// Mitsubishi GX Works2 project: 실린더제어요약   PLC: Q02/Q02H

PROGRAM MAIN
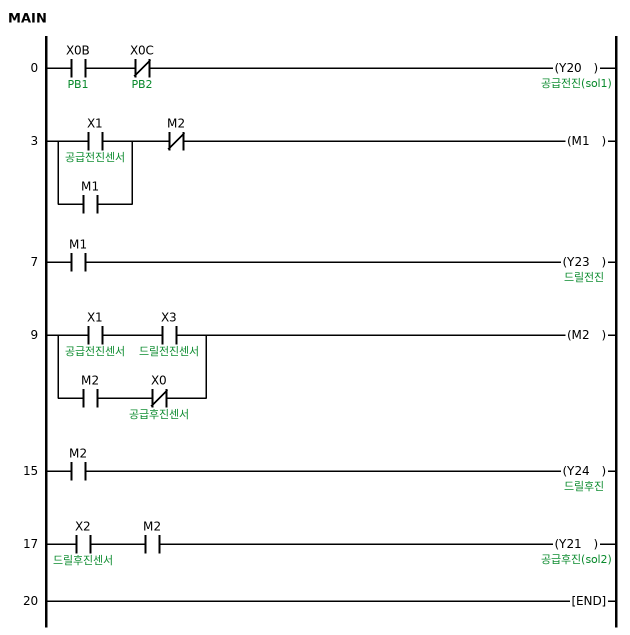
0     LD      X0B  ; PB1
      ANI     X0C  ; PB2
      OUT     Y20  ; 공급전진(sol1)
3     LD      X1  ; 공급전진센서
      OR      M1
      ANI     M2
      OUT     M1
7     LD      M1
      OUT     Y23  ; 드릴전진
9     LD      X1  ; 공급전진센서
      AND     X3  ; 드릴전진센서
      LD      M2
      ANI     X0  ; 공급후진센서
      ORB
      OUT     M2
15    LD      M2
      OUT     Y24  ; 드릴후진
17    LD      X2  ; 드릴후진센서
      AND     M2
      OUT     Y21  ; 공급후진(sol2)
20    END
END_PROGRAM

// device comments not shown above
X4  ; 송출후진센서
X5  ; 송출전진센서
X0D  ; PB3
Y26  ; 송출전진(sol3)
Y27  ; 송출후진(sol4)
